Staubli VAL3: oGripCmd2.pgx

public program oGripCmd2(num nState (dimensions=1))
begin
  dioSet(oGripCmd2,nState)
end
